// Mitsubishi GX Works2 project: CC-Link+ethernet   PLC: Q03UDV

PROGRAM MAIN
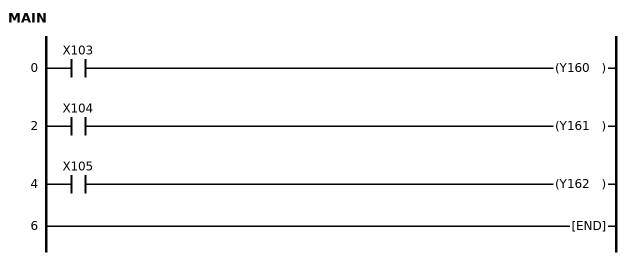
0     LD      X103
      OUT     Y160
2     LD      X104
      OUT     Y161
4     LD      X105
      OUT     Y162
6     END
END_PROGRAM
